(* PLC project CoDeSys External Library Template, WAGO e!COCKPIT e!COCKPIT, author 3S - Smart Software Solutions GmbH *)
(* stored: creationDateTime 2019-10-29T12:37:19.6361823, version 3.5.5.30, modificationDateTime 2019-10-29T12:36:39.3744516, organization 3S - Smart Software Solutions GmbH *)
(* Library project template with all possible element types, docu and a sample project structure *)

FUNCTION_BLOCK fbModbusOdczytZapis
  VAR_INPUT
    intModbusOdczytZapisZadanieRozmiar : INT;  (* Rozmiar tablicy danych modbusa *)
    xOdczytajRejestr : BOOL;  (* Żądanie odczytania rejestru *)
    bAdresOdczyt : BYTE := 2#101000;  (* Adres urządzenia, z którego ma zostać dokonany odczyt *)
    uiAdresRejestruOdczyt : UINT := 2010;  (* Adres rejestru, z którego ma zostać dokonany odczyt *)
    xZapiszRejestr : BOOL;  (* Żądanie zapisania rejestru *)
    bAdresZapis : BYTE;  (* Adres urządzenia, na który ma zostać dokonany zapis *)
    uiAdresRejestruZapis : UINT;  (* Adres rejestru, na który ma zostać dokonany zapis *)
    wZawartoscRejestruZapis : WORD;  (* Dane do zapisu *)
  END_VAR
  VAR_IN_OUT
    arModbusOdczytCykliczny : ARRAY[1..5000] OF typModbusOdczytCykliczny;
    arModbusOdczytZapisZadanie : ARRAY[1..1000] OF typModbusOdczytZapisZadanie;
    intModbusOdczytZapisZadanieZnacznikZapisu : INT;
  END_VAR
  VAR
    tMinimalnyCzasRaportowania : TIME := TIME#15s0ms;
    intPetlaPierwszySkan : INT := 1;
    wZawartoscRejestruOdczyt : WORD;  (* Zawartość odczytanego rejestru *)
    xPierwszyCykl : BOOL := TRUE;  (* Pierwszy cykl programu *)
  END_VAR

            (*			
Autor:					Artur Wyszomirski, 2019-10-11 
Prawa majątkowe: 		Solwena Sp. z o.o., 
Aktualizacje:			2019-10-22: - dodanie wyszukiwania wolnego miejsca w tablicy arModbusOdczytCykliczny
									- wprowadzenie domyślnych wartości dla bAdresOdczyt i uiAdresRejestruOdczyt
									- przypisywanie wartości ltCzestotliwosc i pZmiennaReferencyjna w pierwszym cyklu programu

Opis:					Odczyt i zapis dowolnego rejestru Modbus				
*)

// Pierwszy cykl programu
IF xPierwszyCykl THEN
	WHILE arModbusOdczytCykliczny[intPetlaPierwszySkan].bAdresUrzadzenia <> 0 DO
		intPetlaPierwszySkan := intPetlaPierwszySkan + 1;
	END_WHILE
END_IF

// Odczyt
IF xPierwszyCykl THEN
	arModbusOdczytCykliczny[intPetlaPierwszySkan].ltCzestotliwosc := TIME_TO_LTIME(tMinimalnyCzasRaportowania);
	arModbusOdczytCykliczny[intPetlaPierwszySkan].pZmiennaReferencyjna := ADR(wZawartoscRejestruOdczyt);
END_IF
IF xOdczytajRejestr OR xPierwszyCykl THEN
	arModbusOdczytCykliczny[intPetlaPierwszySkan].bAdresUrzadzenia := bAdresOdczyt;
	arModbusOdczytCykliczny[intPetlaPierwszySkan].bFunkcja := TO_BYTE(enumModbusKodyFunkcji.OdczytNRejestrow);
	arModbusOdczytCykliczny[intPetlaPierwszySkan].uiAdresRejestru := uiAdresRejestruOdczyt;

END_IF

// Zapis
IF xZapiszRejestr THEN
	fnModbusZapisRejestru(	bAdresUrzadzenia := bAdresZapis,
							bFunkcja := INT_TO_BYTE(enumModbusKodyFunkcji.ZapisRejestru),
							uiAdresRejestru := uiAdresRejestruZapis,
							pZmiennaReferencyjna := 0,
							wWartoscDoZapisania := wZawartoscRejestruZapis,
							intModbusOdczytZapisZadanieRozmiar := intModbusOdczytZapisZadanieRozmiar,
							arModbusOdczytZapisZadanie := arModbusOdczytZapisZadanie,
							intModbusOdczytZapisZadanieZnacznikZapisu := intModbusOdczytZapisZadanieZnacznikZapisu);
END_IF
	
xPierwszyCykl := FALSE;
          
END_FUNCTION_BLOCK
